// TIA Portal V17 export
// export: Created 2024-08-20T13:37:00.4220976Z, ExportSetting WithDefaults, DisplayName Totally Integrated Automation Portal, DisplayVersion V17 Update 4, DisplayName TIA Portal Openness, DisplayVersion V17 Update 4, DisplayName TIA Portal Version Control Interface, DisplayVersion V17, DisplayName STEP 7 Professional, DisplayVersion V17 Update 4, DisplayName STEP 7 Safety, DisplayVersion V17, DisplayName WinCC Advanced, DisplayVersion V17 Update 4
FUNCTION_BLOCK "ANALOGICOS"   // FB101, LAD
{ S7_Optimized_Access := 'FALSE' }
VERSION : 0.1
// stored: AutoNumber false, IsIECCheckEnabled false, SetENOAutomatically false, UDAEnableTagReadback false
   VAR
      LIT_001 { S7_SetPoint := 'True'} : "INSTRUMENTO";   // Nível Tanque
   END_VAR
BEGIN

REGION Network 1: Nível Tanque (Sensor tipo radar)
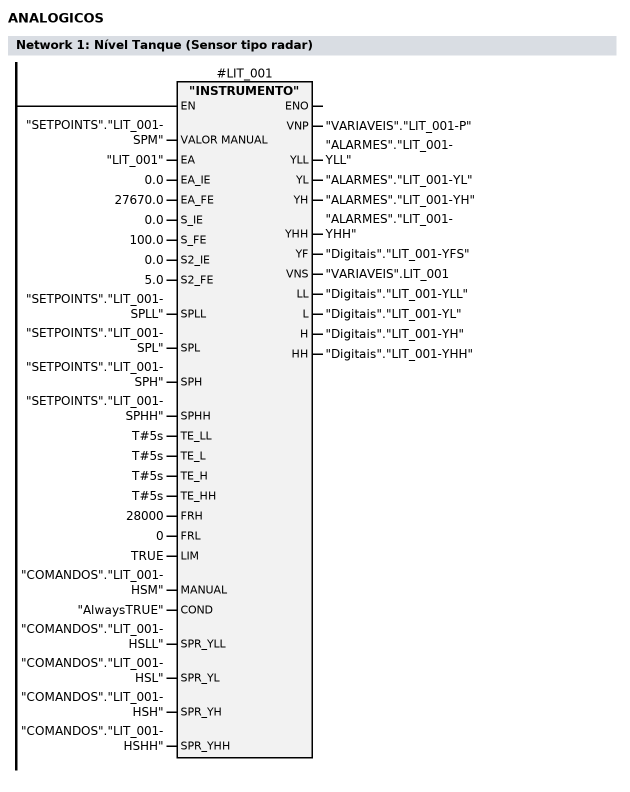
   RUNG wire#powerrail
      #LIT_001("VALOR MANUAL" := "SETPOINTS"."LIT_001-SPM", EA := "LIT_001", EA_IE := 0.0, EA_FE := 27670.0, S_IE := 0.0, S_FE := 100.0, S2_IE := 0.0, S2_FE := 5.0, SPLL := "SETPOINTS"."LIT_001-SPLL", SPL := "SETPOINTS"."LIT_001-SPL", SPH := "SETPOINTS"."LIT_001-SPH", SPHH := "SETPOINTS"."LIT_001-SPHH", TE_LL := T#5s, TE_L := T#5s, TE_H := T#5s, TE_HH := T#5s, FRH := 28000, FRL := 0, LIM := TRUE, MANUAL := "COMANDOS"."LIT_001-HSM", COND := "AlwaysTRUE", SPR_YLL := "COMANDOS"."LIT_001-HSLL", SPR_YL := "COMANDOS"."LIT_001-HSL", SPR_YH := "COMANDOS"."LIT_001-HSH", SPR_YHH := "COMANDOS"."LIT_001-HSHH", VNP => "VARIAVEIS"."LIT_001-P", YLL => "ALARMES"."LIT_001-YLL", YL => "ALARMES"."LIT_001-YL", YH => "ALARMES"."LIT_001-YH", YHH => "ALARMES"."LIT_001-YHH", YF => "Digitais"."LIT_001-YFS", VNS => "VARIAVEIS".LIT_001, LL => "Digitais"."LIT_001-YLL", L => "Digitais"."LIT_001-YL", H => "Digitais"."LIT_001-YH", HH => "Digitais"."LIT_001-YHH")
   END_RUNG
   // the same network as SCL:
   #LIT_001("VALOR MANUAL" := "SETPOINTS"."LIT_001-SPM",   // "INSTRUMENTO"
            EA := "LIT_001",
            EA_IE := 0.0,
            EA_FE := 27670.0,
            S_IE := 0.0,
            S_FE := 100.0,
            S2_IE := 0.0,
            S2_FE := 5.0,
            SPLL := "SETPOINTS"."LIT_001-SPLL",
            SPL := "SETPOINTS"."LIT_001-SPL",
            SPH := "SETPOINTS"."LIT_001-SPH",
            SPHH := "SETPOINTS"."LIT_001-SPHH",
            TE_LL := T#5s,
            TE_L := T#5s,
            TE_H := T#5s,
            TE_HH := T#5s,
            FRH := 28000,
            FRL := 0,
            LIM := TRUE,
            MANUAL := "COMANDOS"."LIT_001-HSM",
            COND := "AlwaysTRUE",
            SPR_YLL := "COMANDOS"."LIT_001-HSLL",
            SPR_YL := "COMANDOS"."LIT_001-HSL",
            SPR_YH := "COMANDOS"."LIT_001-HSH",
            SPR_YHH := "COMANDOS"."LIT_001-HSHH",
            VNP => "VARIAVEIS"."LIT_001-P",
            YLL => "ALARMES"."LIT_001-YLL",
            YL => "ALARMES"."LIT_001-YL",
            YH => "ALARMES"."LIT_001-YH",
            YHH => "ALARMES"."LIT_001-YHH",
            YF => "Digitais"."LIT_001-YFS",
            VNS => "VARIAVEIS".LIT_001,
            LL => "Digitais"."LIT_001-YLL",
            L => "Digitais"."LIT_001-YL",
            H => "Digitais"."LIT_001-YH",
            HH => "Digitais"."LIT_001-YHH");
END_REGION
END_FUNCTION_BLOCK
